FUNCTION_BLOCK StatusInfo (* Composite Function Block Type *)
  (* Standard: 61499-2 *)
  (* Version 0.0, 3/4/2026, Schneider Electric, template *)
  PACKAGE SE.Nereda;
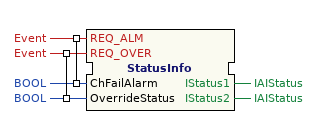
  EVENT_INPUT
    REQ_ALM WITH ChFailAlarm;
    REQ_OVER WITH OverrideStatus;
  END_EVENT
  VAR_INPUT
    ChFailAlarm : BOOL;
    OverrideStatus : BOOL;
  END_VAR
  PLUGS
    IStatus1 : IAIStatus;
    IStatus2 : IAIStatus;
  END_PLUGS
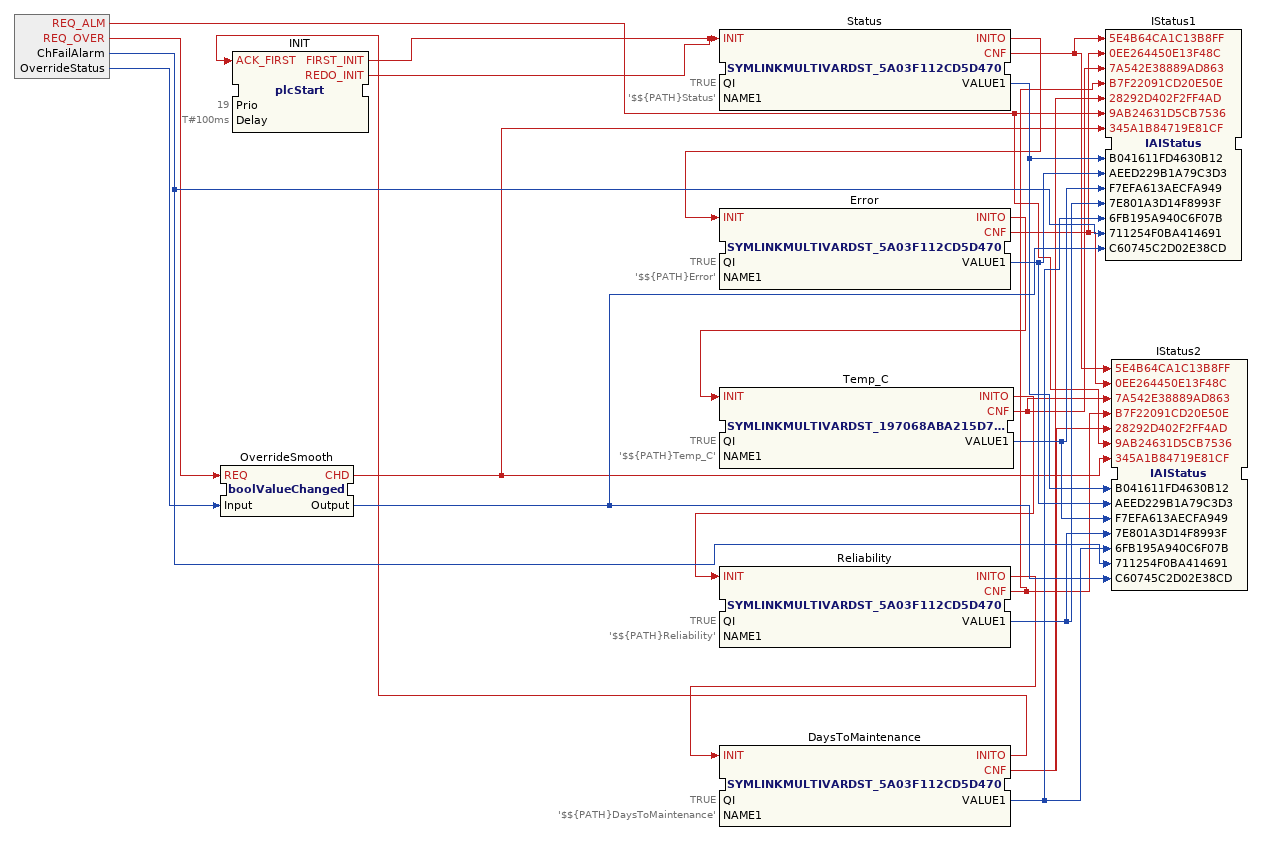
  (* 03 - FIELD INTERFACE IN *)
  (* 02 - FUNCTIONNAL OUTPUT INTERFACE *)
  (* 00 - INITIALIZATION *)
  (* 01 - FUNCTIONNAL INPUT INTERFACE *)
  FBS
    Status : SYMLINKMULTIVARDST_5A03F112CD5D470(QI := TRUE, NAME1 := '$${PATH}Status'); {SET_ATTRIBUTE(Configuration.GenericFBType.InterfaceParams, Runtime.System#I:=1;VALUE${I$}:INT)}
    Temp_C : SYMLINKMULTIVARDST_197068ABA215D7EBA(QI := TRUE, NAME1 := '$${PATH}Temp_C'); {SET_ATTRIBUTE(Configuration.GenericFBType.InterfaceParams, Runtime.System#I:=1;VALUE${I$}:REAL)}
    Error : SYMLINKMULTIVARDST_5A03F112CD5D470(QI := TRUE, NAME1 := '$${PATH}Error'); {SET_ATTRIBUTE(Configuration.GenericFBType.InterfaceParams, Runtime.System#I:=1;VALUE${I$}:INT)}
    Reliability : SYMLINKMULTIVARDST_5A03F112CD5D470(QI := TRUE, NAME1 := '$${PATH}Reliability'); {SET_ATTRIBUTE(Configuration.GenericFBType.InterfaceParams, Runtime.System#I:=1;VALUE${I$}:INT)}
    DaysToMaintenance : SYMLINKMULTIVARDST_5A03F112CD5D470(QI := TRUE, NAME1 := '$${PATH}DaysToMaintenance'); {SET_ATTRIBUTE(Configuration.GenericFBType.InterfaceParams, Runtime.System#I:=1;VALUE${I$}:INT)}
    INIT : plcStart(Prio := 19, Delay := T#100ms);
    OverrideSmooth : boolValueChanged;
  END_FBS
  EVENT_CONNECTIONS
    Error.INITO TO Temp_C.INIT;
    Temp_C.INITO TO Reliability.INIT;
    Reliability.INITO TO DaysToMaintenance.INIT;
    Status.INITO TO Error.INIT;
    INIT.FIRST_INIT TO Status.INIT;
    INIT.REDO_INIT TO Status.INIT;
    DaysToMaintenance.INITO TO INIT.ACK_FIRST;
    Status.CNF TO IStatus1.5E4B64CA1C13B8FF;
    Status.CNF TO IStatus2.5E4B64CA1C13B8FF;
    Error.CNF TO IStatus1.0EE264450E13F48C;
    Error.CNF TO IStatus2.0EE264450E13F48C;
    Temp_C.CNF TO IStatus2.7A542E38889AD863;
    Temp_C.CNF TO IStatus1.7A542E38889AD863;
    Reliability.CNF TO IStatus1.B7F22091CD20E50E;
    Reliability.CNF TO IStatus2.B7F22091CD20E50E;
    DaysToMaintenance.CNF TO IStatus1.28292D402F2FF4AD;
    DaysToMaintenance.CNF TO IStatus2.28292D402F2FF4AD;
    REQ_ALM TO IStatus1.9AB24631D5CB7536;
    REQ_ALM TO IStatus2.9AB24631D5CB7536;
    OverrideSmooth.CHD TO IStatus1.345A1B84719E81CF;
    OverrideSmooth.CHD TO IStatus2.345A1B84719E81CF;
    REQ_OVER TO OverrideSmooth.REQ;
  END_CONNECTIONS
  DATA_CONNECTIONS
    Status.VALUE1 TO IStatus1.B041611FD4630B12;
    Status.VALUE1 TO IStatus2.B041611FD4630B12;
    Error.VALUE1 TO IStatus1.AEED229B1A79C3D3;
    Error.VALUE1 TO IStatus2.AEED229B1A79C3D3;
    Temp_C.VALUE1 TO IStatus1.F7EFA613AECFA949;
    Temp_C.VALUE1 TO IStatus2.F7EFA613AECFA949;
    Reliability.VALUE1 TO IStatus1.7E801A3D14F8993F;
    Reliability.VALUE1 TO IStatus2.7E801A3D14F8993F;
    DaysToMaintenance.VALUE1 TO IStatus1.6FB195A940C6F07B;
    DaysToMaintenance.VALUE1 TO IStatus2.6FB195A940C6F07B;
    ChFailAlarm TO IStatus1.711254F0BA414691;
    ChFailAlarm TO IStatus2.711254F0BA414691;
    OverrideSmooth.Output TO IStatus1.C60745C2D02E38CD;
    OverrideSmooth.Output TO IStatus2.C60745C2D02E38CD;
    OverrideStatus TO OverrideSmooth.Input;
  END_CONNECTIONS
END_FUNCTION_BLOCK
